(* CODESYS project sys time and date_RECOVERED_2026-08-13T11-07-18.project

Project tree, tasks and I/O mapping:
  Device : CODESYS Control Win V3 x64, CODESYS, version 3.5.22.30
    application Application
      libraries: Standard, 3.5.22.0 (System); SysTime, 3.5.17.0 (System); SysTypes Interfaces, * (System)
      task MainTask (cyclic, interval t#20ms, priority 1) calls PLC_PRG
      program PLC_PRG [LD]
*)

// Device/Application/PLC_PRG
PROGRAM PLC_PRG
VAR
END_VAR

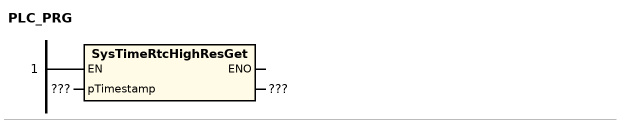
// NETWORK 1
SysTimeRtcHighResGet();

END_PROGRAM
